FUNCTION_BLOCK MockCyclic IMPLEMENTS I_Cyclic, I_Object
VAR
	_isRegistered : BOOL;
END_VAR

METHOD Cycle : HRESULT
END_METHOD

METHOD IsRegistered : BOOL
VAR_INPUT
END_VAR
IsRegistered := _isRegistered;
END_METHOD

METHOD RegisterWithParent
VAR_INPUT
	Parent	: I_HostObjects;
END_VAR
IF NOT _isRegistered THEN
	IF SUCCEEDED( Parent.RegisterCyclic(THIS^)) THEN
		_isRegistered := TRUE;
	ELSE
		_isRegistered := FALSE;
	END_IF
END_IF
END_METHOD

END_FUNCTION_BLOCK

(* stored: Version 1.1.0.1
   POU MockCyclic: Id {459c9319-db86-4d6a-b774-a97d62f0aee0}, SpecialFunc None
   Method Cycle: Id {2fdaa782-1cce-42d3-b0fd-0a553501ea73}
   Method IsRegistered: Id {432ff809-df19-4dfc-b853-62c50ce79958}
   Method RegisterWithParent: Id {53309e55-7b39-4961-93ff-498d9c30e110} *)
